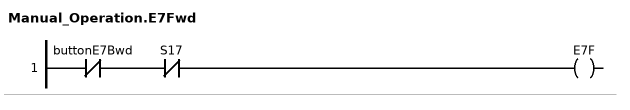
[picture p24: Manual_Operation.E7Fwd (LD)]
_LD_ (* Ladder Diagram *)
NETWORK 1
	[/buttonE7Bwd] - [/S17] --- (E7F)
_END_LD_
(* the same logic as Structured Text *)
(* Network 1 *)
E7F := NOT buttonE7Bwd AND NOT S17;
END_ACTION
ACTION E8Bwd:
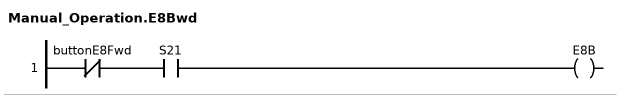
_LD_ (* Ladder Diagram *)
NETWORK 1
	[/buttonE8Fwd] - [S21] --- (E8B)
_END_LD_
(* the same logic as Structured Text *)
(* Network 1 *)
E8B := NOT buttonE8Fwd AND S21;
END_ACTION

(* POU Automatic_Operation, SFC *)
PROGRAM Automatic_Operation
VAR
END_VAR
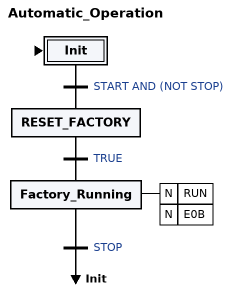
INITIAL_STEP Init:
END_STEP
TRANSITION FROM Init TO RESET_FACTORY := START AND (NOT STOP);
END_TRANSITION
STEP RESET_FACTORY:
END_STEP
TRANSITION FROM RESET_FACTORY TO Factory_Running := TRUE;
END_TRANSITION
STEP Factory_Running:
	RUN(N);
	E0B(N);
END_STEP
TRANSITION FROM Factory_Running TO Init := STOP;
END_TRANSITION
END_PROGRAM

(* POU Lobby, SFC *)
PROGRAM Lobby
VAR
	LOBBY_DELIVER: BOOL;		(*Deliver from lobby to roof*)
END_VAR
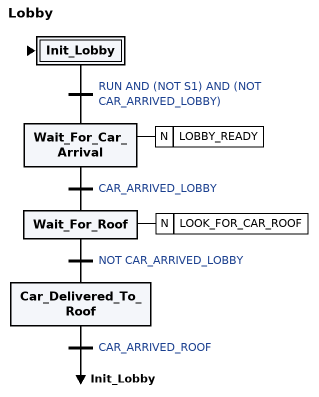
INITIAL_STEP Init_Lobby:
END_STEP
TRANSITION FROM Init_Lobby TO Wait_For_Car_Arrival := RUN AND (NOT S1) AND (NOT CAR_ARRIVED_LOBBY);
END_TRANSITION
STEP Wait_For_Car_Arrival:
	LOBBY_READY(N);
END_STEP
TRANSITION FROM Wait_For_Car_Arrival TO Wait_For_Roof := CAR_ARRIVED_LOBBY;
END_TRANSITION
STEP Wait_For_Roof:
	LOOK_FOR_CAR_ROOF(N);
END_STEP
TRANSITION FROM Wait_For_Roof TO Car_Delivered_To_Roof := NOT CAR_ARRIVED_LOBBY;
END_TRANSITION
STEP Car_Delivered_To_Roof:
END_STEP
TRANSITION FROM Car_Delivered_To_Roof TO Init_Lobby := CAR_ARRIVED_ROOF;
END_TRANSITION
END_PROGRAM

(* POU Roof, SFC *)
PROGRAM Roof
VAR
	Roof_Fwd_Go: BOOL;
	Temp_Var_Roof: BOOL;
	LOBBY_DELIVER: BOOL; (*Doesn't do anything rn*)
END_VAR
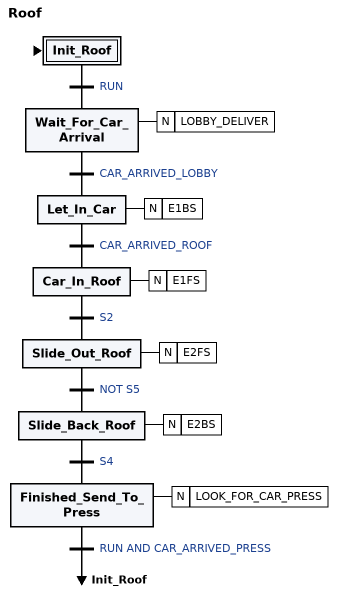
INITIAL_STEP Init_Roof:
END_STEP
TRANSITION FROM Init_Roof TO Wait_For_Car_Arrival := RUN;
END_TRANSITION
STEP Wait_For_Car_Arrival:
	LOBBY_DELIVER(N);
END_STEP
TRANSITION FROM Wait_For_Car_Arrival TO Let_In_Car := CAR_ARRIVED_LOBBY;
END_TRANSITION
STEP Let_In_Car:
	E1BS(N);
END_STEP
TRANSITION FROM Let_In_Car TO Car_In_Roof := CAR_ARRIVED_ROOF;
END_TRANSITION
STEP Car_In_Roof:
	E1FS(N);
END_STEP
TRANSITION FROM Car_In_Roof TO Slide_Out_Roof := S2;
END_TRANSITION
STEP Slide_Out_Roof:
	E2FS(N);
END_STEP
TRANSITION FROM Slide_Out_Roof TO Slide_Back_Roof := NOT S5;
END_TRANSITION
STEP Slide_Back_Roof:
	E2BS(N);
END_STEP
TRANSITION FROM Slide_Back_Roof TO Finished_Send_To_Press := S4;
END_TRANSITION
STEP Finished_Send_To_Press:
	LOOK_FOR_CAR_PRESS(N);
END_STEP
TRANSITION FROM Finished_Send_To_Press TO Init_Roof := RUN AND CAR_ARRIVED_PRESS;
END_TRANSITION
END_PROGRAM

(* POU Press, SFC *)
PROGRAM Press
VAR
END_VAR
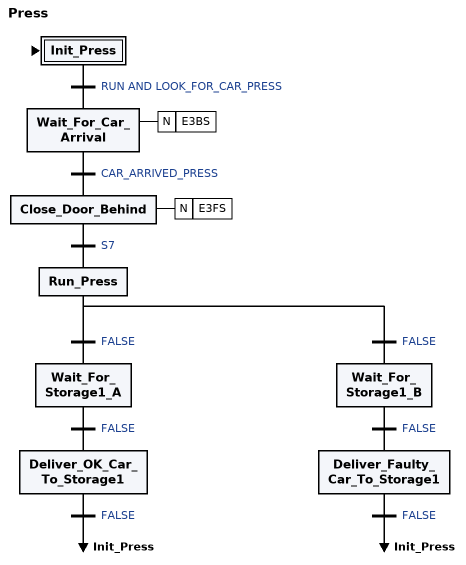
INITIAL_STEP Init_Press:
END_STEP
TRANSITION FROM Init_Press TO Wait_For_Car_Arrival := RUN AND LOOK_FOR_CAR_PRESS;
END_TRANSITION
STEP Wait_For_Car_Arrival:
	E3BS(N);
END_STEP
TRANSITION FROM Wait_For_Car_Arrival TO Close_Door_Behind := CAR_ARRIVED_PRESS;
END_TRANSITION
STEP Close_Door_Behind:
	E3FS(N);
END_STEP
TRANSITION FROM Close_Door_Behind TO Run_Press := S7;
END_TRANSITION
STEP Run_Press:
END_STEP
TRANSITION FROM Run_Press TO Wait_For_Storage1_A := FALSE;
END_TRANSITION
TRANSITION FROM Run_Press TO Wait_For_Storage1_B := FALSE;
END_TRANSITION
STEP Wait_For_Storage1_A:
END_STEP
TRANSITION FROM Wait_For_Storage1_A TO Deliver_OK_Car_To_Storage1 := FALSE;
END_TRANSITION
STEP Wait_For_Storage1_B:
END_STEP
TRANSITION FROM Wait_For_Storage1_B TO Deliver_Faulty_Car_To_Storage1 := FALSE;
END_TRANSITION
STEP Deliver_Faulty_Car_To_Storage1:
END_STEP
TRANSITION FROM Deliver_Faulty_Car_To_Storage1 TO Init_Press := FALSE;
END_TRANSITION
STEP Deliver_OK_Car_To_Storage1:
END_STEP
TRANSITION FROM Deliver_OK_Car_To_Storage1 TO Init_Press := FALSE;
END_TRANSITION
END_PROGRAM

(* POU Storage1, SFC *)
PROGRAM Storage1
VAR
END_VAR
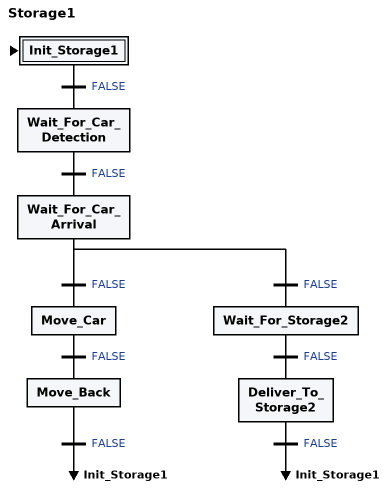
INITIAL_STEP Init_Storage1:
END_STEP
TRANSITION FROM Init_Storage1 TO Wait_For_Car_Detection := FALSE;
END_TRANSITION
STEP Wait_For_Car_Detection:
END_STEP
TRANSITION FROM Wait_For_Car_Detection TO Wait_For_Car_Arrival := FALSE;
END_TRANSITION
STEP Wait_For_Car_Arrival:
END_STEP
TRANSITION FROM Wait_For_Car_Arrival TO Move_Car := FALSE;
END_TRANSITION
TRANSITION FROM Wait_For_Car_Arrival TO Wait_For_Storage2 := FALSE;
END_TRANSITION
STEP Move_Car:
END_STEP
TRANSITION FROM Move_Car TO Move_Back := FALSE;
END_TRANSITION
STEP Move_Back:
END_STEP
TRANSITION FROM Move_Back TO Init_Storage1 := FALSE;
END_TRANSITION
STEP Wait_For_Storage2:
END_STEP
TRANSITION FROM Wait_For_Storage2 TO Deliver_To_Storage2 := FALSE;
END_TRANSITION
STEP Deliver_To_Storage2:
END_STEP
TRANSITION FROM Deliver_To_Storage2 TO Init_Storage1 := FALSE;
END_TRANSITION
END_PROGRAM

(* POU Storage2, SFC *)
PROGRAM Storage2
VAR
END_VAR
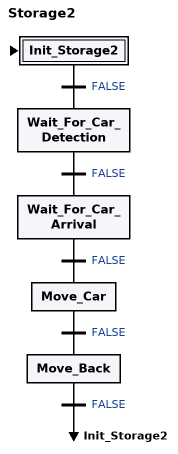
INITIAL_STEP Init_Storage2:
END_STEP
TRANSITION FROM Init_Storage2 TO Wait_For_Car_Detection := FALSE;
END_TRANSITION
STEP Wait_For_Car_Detection:
END_STEP
TRANSITION FROM Wait_For_Car_Detection TO Wait_For_Car_Arrival := FALSE;
END_TRANSITION
STEP Wait_For_Car_Arrival:
END_STEP
TRANSITION FROM Wait_For_Car_Arrival TO Move_Car := FALSE;
END_TRANSITION
STEP Move_Car:
END_STEP
TRANSITION FROM Move_Car TO Move_Back := FALSE;
END_TRANSITION
STEP Move_Back:
END_STEP
TRANSITION FROM Move_Back TO Init_Storage2 := FALSE;
END_TRANSITION
END_PROGRAM

(* POU Automatic_Conditional, LD *)
PROGRAM Automatic_Conditional
VAR
	T0: TON;		(*Timer utanför roof*)
	T3: TON;
	T6: TON;
	T9: TON;
	T14: TON; (*Kan behöva tweak:as*)
	T19: TON;
END_VAR
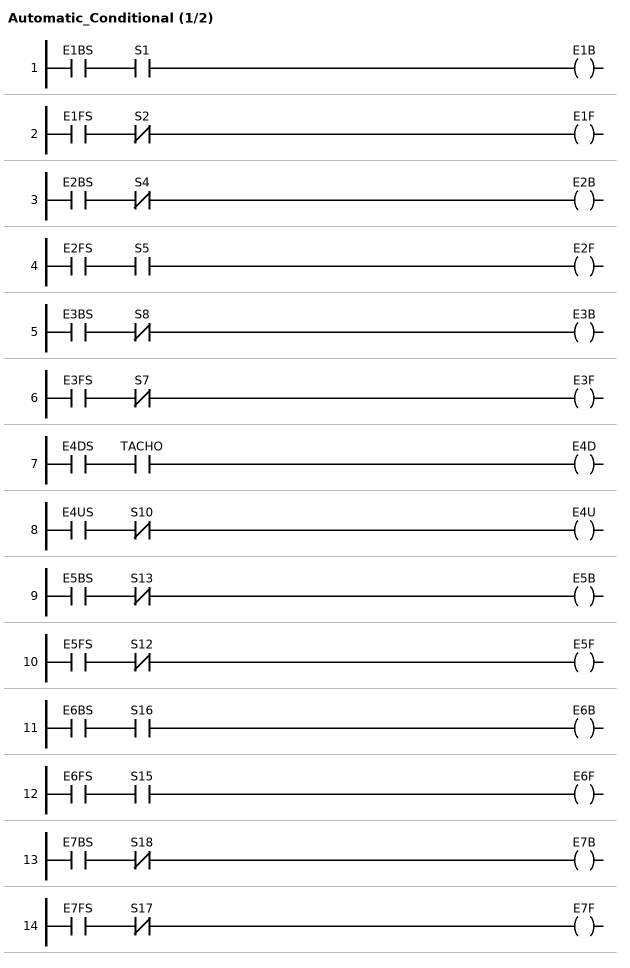
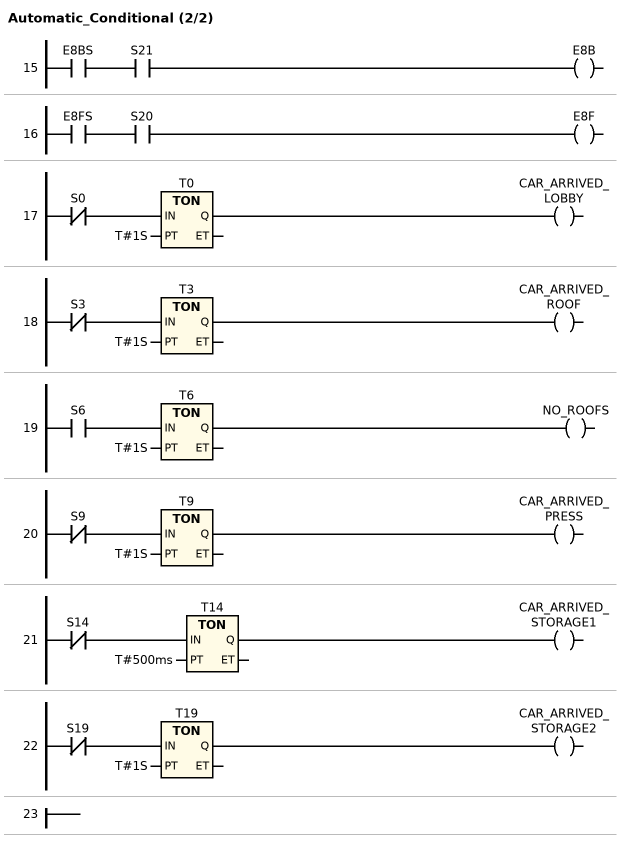
_LD_ (* Ladder Diagram *)
NETWORK 1
	[E1BS] - [S1] --- (E1B)
NETWORK 2
	[E1FS] - [/S2] --- (E1F)
NETWORK 3
	[E2BS] - [/S4] --- (E2B)
NETWORK 4
	[E2FS] - [S5] --- (E2F)
NETWORK 5
	[E3BS] - [/S8] --- (E3B)
NETWORK 6
	[E3FS] - [/S7] --- (E3F)
NETWORK 7
	[E4DS] - [TACHO] --- (E4D)
NETWORK 8
	[E4US] - [/S10] --- (E4U)
NETWORK 9
	[E5BS] - [/S13] --- (E5B)
NETWORK 10
	[E5FS] - [/S12] --- (E5F)
NETWORK 11
	[E6BS] - [S16] --- (E6B)
NETWORK 12
	[E6FS] - [S15] --- (E6F)
NETWORK 13
	[E7BS] - [/S18] --- (E7B)
NETWORK 14
	[E7FS] - [/S17] --- (E7F)
NETWORK 15
	[E8BS] - [S21] --- (E8B)
NETWORK 16
	[E8FS] - [S20] --- (E8F)
NETWORK 17
	[/S0] - T0:TON(IN: *, PT: T#1S) --- (CAR_ARRIVED_LOBBY)
NETWORK 18
	[/S3] - T3:TON(IN: *, PT: T#1S) --- (CAR_ARRIVED_ROOF)
NETWORK 19
	[S6] - T6:TON(IN: *, PT: T#1S) --- (NO_ROOFS)
NETWORK 20
	[/S9] - T9:TON(IN: *, PT: T#1S) --- (CAR_ARRIVED_PRESS)
NETWORK 21
	[/S14] - T14:TON(IN: *, PT: T#500ms) --- (CAR_ARRIVED_STORAGE1)
NETWORK 22
	[/S19] - T19:TON(IN: *, PT: T#1S) --- (CAR_ARRIVED_STORAGE2)
NETWORK 23
	*
_END_LD_
(* the same logic as Structured Text *)
(* Network 1 *)
E1B := E1BS AND S1;
(* Network 2 *)
E1F := E1FS AND NOT S2;
(* Network 3 *)
E2B := E2BS AND NOT S4;
(* Network 4 *)
E2F := E2FS AND S5;
(* Network 5 *)
E3B := E3BS AND NOT S8;
(* Network 6 *)
E3F := E3FS AND NOT S7;
(* Network 7 *)
E4D := E4DS AND TACHO;
(* Network 8 *)
E4U := E4US AND NOT S10;
(* Network 9 *)
E5B := E5BS AND NOT S13;
(* Network 10 *)
E5F := E5FS AND NOT S12;
(* Network 11 *)
E6B := E6BS AND S16;
(* Network 12 *)
E6F := E6FS AND S15;
(* Network 13 *)
E7B := E7BS AND NOT S18;
(* Network 14 *)
E7F := E7FS AND NOT S17;
(* Network 15 *)
E8B := E8BS AND S21;
(* Network 16 *)
E8F := E8FS AND S20;
(* Network 17 *)
T0(IN := NOT S0, PT := T#1S);
CAR_ARRIVED_LOBBY := T0.Q;
(* Network 18 *)
T3(IN := NOT S3, PT := T#1S);
CAR_ARRIVED_ROOF := T3.Q;
(* Network 19 *)
T6(IN := S6, PT := T#1S);
NO_ROOFS := T6.Q;
(* Network 20 *)
T9(IN := NOT S9, PT := T#1S);
CAR_ARRIVED_PRESS := T9.Q;
(* Network 21 *)
T14(IN := NOT S14, PT := T#500ms);
CAR_ARRIVED_STORAGE1 := T14.Q;
(* Network 22 *)
T19(IN := NOT S19, PT := T#1S);
CAR_ARRIVED_STORAGE2 := T19.Q;
(* Network 23 *)
END_PROGRAM
